TYPE stTarget2D EXTENDS stTarget :
STRUCT
	pose : stPose2D;
END_STRUCT
END_TYPE

(* stored: Version 1.1.0.1, ProductVersion 3.1.4026.18
   DUT stTarget2D: Id {c1b2c3d4-3333-3333-3333-333333333333} *)
